(*

short summary
=============

.. <legal notes>

legal notes
=================
| SPDX-FileCopyrightText: © 2023 ekvip automation GmbH <info@ekvip.de>
| SPDX-License-Identifier: Apache-2.0
| For details check: Apache-2.0_

.. _Apache-2.0: https://www.apache.org/licenses/LICENSE-2.0

.. </legal notes>

*)

{warning 'header is generated please add your documentation'}
TYPE IsLengthBasicData :
STRUCT
	StringToTest	: STRING;
	WStringToTest	: WSTRING;
	ExpectedResult  : BOOL;
	ExpectedLength	: UDINT; 
	FuncType		: FunctionType;
	typeToTest      : TypeToTest;  	
END_STRUCT
END_TYPE

(* stored: Version 1.1.0.1, ProductVersion 3.1.4024.12
   DUT IsLengthBasicData: Id {0a4e04e4-2c88-49e5-849e-f7bc8fcbad2e} *)
